// Mitsubishi GX Works2 project: 인터록회로   PLC: Q02/Q02H

PROGRAM MAIN
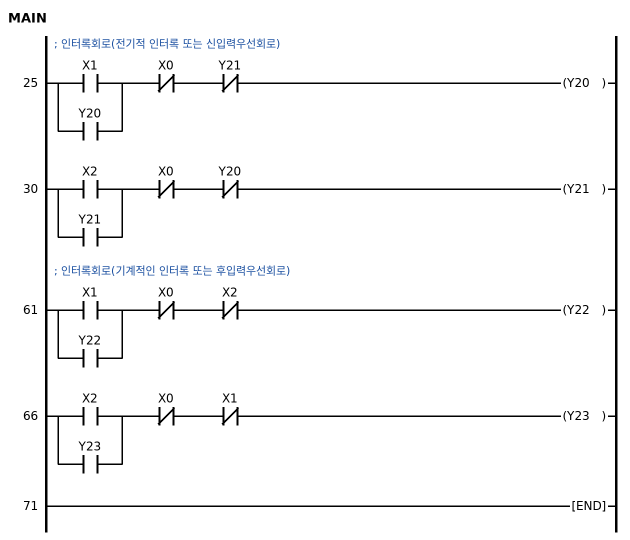
; 인터록회로(전기적 인터록 또는 신입력우선회로)
25    LD      X1
      OR      Y20
      ANI     X0
      ANI     Y21
      OUT     Y20
30    LD      X2
      OR      Y21
      ANI     X0
      ANI     Y20
      OUT     Y21
; 인터록회로(기계적인 인터록 또는 후입력우선회로)
61    LD      X1
      OR      Y22
      ANI     X0
      ANI     X2
      OUT     Y22
66    LD      X2
      OR      Y23
      ANI     X0
      ANI     X1
      OUT     Y23
71    END
END_PROGRAM
